// TwinCAT 3 PLC project HelloWorld
// ProgramVersion: 3.1.4024.0
// libraries:
//   Tc2_Standard, * (Beckhoff Automation GmbH)
//   Tc2_System, * (Beckhoff Automation GmbH)
//   Tc2_Utilities, * (Beckhoff Automation GmbH)
//   Tc3_Module, * (Beckhoff Automation GmbH)
// project tree:
//   DUTs/ E_Color.TcDUT (not stored), E_Event.TcDUT (not stored), ST_Event.TcDUT (not stored), ST_Student.TcDUT (not stored)
//   GVLs/ Nums.TcGVL (not stored)
//   / PlcTask.TcTTO (not stored)
//   POUs/ Celcius_Fahrenheit.TcPOU (not stored), F_Add.TcPOU (not stored), F_InitializeStudentDetails.TcPOU (not stored), F_Loops.TcPOU (not stored), F_Multiply.TcPOU (not stored), F_PrimeCheck.TcPOU (not stored), F_UpdateTimeWithSystemTime.TcPOU (not stored), F_HelloWorld.TcPOU, MAIN.TcPOU, My_Program.TcPOU (not stored)
// real-time tasks:
//   TASK PlcTask: cycle T#10ms, priority 20, ADS port 350

// ---- POUs/F_HelloWorld.TcPOU
FUNCTION F_HelloWorld
VAR_INPUT
END_VAR
VAR
	nNum :DINT := 329;
END_VAR


		ADSLOGSTR(msgCtrlMask := ADSLOG_MSGTYPE_ERROR OR ADSLOG_MSGTYPE_LOG,
			msgFmtStr:= 'Hello world!!',
			strArg:='');
		ADSLOGDINT(msgCtrlMask := ADSLOG_MSGTYPE_WARN, msgFmtStr := 'value of num is %d', dintArg := nNum );

END_FUNCTION

// ---- POUs/MAIN.TcPOU
PROGRAM MAIN
VAR
	fFahrenheit : REAL;
	stEventOne : ST_Event;
	bFlag : BOOL := FALSE;
	nSum : INT;
	nProd : DINT;
	bIsPrime : BOOL;
	nResultFromLoop1 : INT;
	nResultFromLoop2 : INT;
	nResultFromLoop3 : INT;
	nNum1 :INT := 22;
	
	stStudentReference1 : ST_Student;
END_VAR


IF NOT bFlag THEN 
(*fFahrenheit := Celcius_Fahrenheit(fCelcius := 5.0);
F_UpdateTimeWithSystemTime(stEventOne);
F_Add(nFirstNum:= nNum1, nSecondNum:= 32,nResult => nSum );
bFlag := TRUE;
nProd := F_Multiply(123,432);
bIsPrime := F_PrimeCheck(nInputNum := 17 );

F_InitializeStudentDetails(stStudentReference1, 'Kamesh', 1 , 21);

F_Loops(10,nResult1 => nResultFromLoop1, nResult2 => nResultFromLoop2, nResult3 => nResultFromLoop3);
*)
F_HelloWorld();
bFlag := TRUE;
END_IF

END_PROGRAM
